TYPE T_Bool : BOOL; END_TYPE

(* stored: Version 1.1.0.1, ProductVersion 3.1.4024.4
   DUT T_Bool: Id {97bf33e2-ad02-4219-994d-0d8c409fa4c5} *)
